// TwinCAT 3 PLC project PnP_MCgroupCM
// Title: Pick And Place Simple Example with MC Group Coordinated Motion
// Company: Beckhoff Automation GmbH
// Description: Disclaimer This publication contains statements about the suitability of our products for certain areas of application. These statements are based on typical features of our products. The examples shown in this publication are for demonstration purposes only. The information provided herein should not be regarded as specific operation characteristics. It is incumbent on the customer to check and decide whether a product is suitable for use in a particular application. We do not give any warranty that the source code which is made available with this publication is complete or accurate. THE SAMPLE CODE CONTAINED IN THIS PUBLICATION IS PROVIDED “AS IS” WITHOUT WARRANTY OF ANY KIND, EITHER EXPRESSED, IMPLIED OR STATUTORY, INCLUDING WITHOUT LIMITATION, ANY WARRANTY WITH RESPECT TO NON-INFRINGEMENT, FREEDOM FROM PROPRIETARY RIGHTS OF THIRD PARTIES OR FITNESS FOR ANY PARTICULAR PURPOSE. This publication may be changed from time to time without prior notice. No liability is assumed for errors and/or omissions. Our products are described in detail in our data sheets and documentations. Product-specific warnings and cautions must be observed. For the latest version of our data sheets and documentations visit our website (www.beckhoff.de). © Beckhoff Automation GmbH & Co. KG The reproduction, distribution and utilization of this document as well as the communication of its contents to others without express authorization is prohibited. Offenders will be held liable for the payment of damages. All rights reserved in the event of the grant of a patent, utility model or design.
// ProgramVersion: 3.1.4018.1
// libraries:
//   PLCToolbox, * (Beckhoff Automation LLC.)
//   Tc2_MC2, * (Beckhoff Automation GmbH)
//   Tc2_Standard, * (Beckhoff Automation GmbH)
//   Tc2_System, * (Beckhoff Automation GmbH)
//   Tc2_Utilities, * (Beckhoff Automation GmbH)
//   Tc3_EventLogger, * (Beckhoff Automation GmbH)
//   Tc3_McCoordinatedMotion, * (Beckhoff Automation GmbH)
//   Tc3_Module, * (Beckhoff Automation GmbH)
// project tree:
//   DUT/ ST_DwellTime.TcDUT, ST_LineSegment.TcDUT
//   / E_Axis.TcDUT, PlcTask.TcTTO
//   GVLs/ GVL.TcGVL
//   POUs/ FB_AddAllAxes.TcPOU, FB_PowerAll.TcPOU, FB_PreparePath.TcPOU, MAIN.TcPOU
// real-time tasks:
//   TASK PlcTask: cycle T#10ms, priority 20, ADS port 350
//   TASK Worker Task: cycle default, priority 32
// motion (NC):
//   TASK NC-Task 1 SAF: cycle T#2ms, priority 4, ADS port 501
//   TASK NC-Task 1 SVB: cycle T#10ms, priority 8, ADS port 511
//   AXIS X (id 1)
//     OtherSettings: AllowMotionCmdToSlave=true
//     encoder EncType=1
//     drive DrvType=5
//       TimeComp: TaskDelayCycles=1
//     controller CtrType=1
//       CtrPara: PriorControlFactor=1
//         Observer: BandWidth=20
//   AXIS Y (id 2)
//     OtherSettings: AllowMotionCmdToSlave=true
//     encoder EncType=1
//     drive DrvType=5
//       TimeComp: TaskDelayCycles=1
//     controller CtrType=1
//       CtrPara: PriorControlFactor=1
//         Observer: BandWidth=20
// variable links:
//   PnP_MCgroupCM/PnP_MCgroupCM Instance <-> NC-Task 1 SAF/Axes/X
//     PlcTask Inputs/GVL.stAxis[1].NcToPlc <-> Outputs/ToPlc
//     PlcTask Outputs/GVL.stAxis[1].PlcToNc <-> Inputs/FromPlc
//   PnP_MCgroupCM/PnP_MCgroupCM Instance <-> NC-Task 1 SAF/Axes/Y
//     PlcTask Inputs/GVL.stAxis[2].NcToPlc <-> Outputs/ToPlc
//     PlcTask Outputs/GVL.stAxis[2].PlcToNc <-> Inputs/FromPlc
//   PnP_MCgroupCM/PnP_MCgroupCM Instance <-> NC-Task 1 SAF/Objects/Group2 (MC Group Coordinated Motion)
//     PlcTask Inputs/GVL.stGroupRef.NcToPlc <-> Group Outputs/ToPLC
//     PlcTask Outputs/GVL.stGroupRef.PlcToNc <-> Group Inputs/FromPLC

CONFIGURATION PnP_MCgroupCM
    RESOURCE PLC ON TwinCAT3
        TASK PlcTask(INTERVAL := T#10ms, PRIORITY := 20);
        PROGRAM MAIN WITH PlcTask : MAIN;
    END_RESOURCE
END_CONFIGURATION

// ---- DUT/ST_DwellTime.TcDUT
TYPE ST_DwellTime :
STRUCT
	DwellTime	: TIME;
	BufferMode	: MC_BUFFER_MODE := mcBuffered;
	InvokeId	: UDINT;
END_STRUCT
END_TYPE

// ---- DUT/ST_LineSegment.TcDUT
TYPE
ST_LineSegment :
STRUCT
	TargetPos					: ARRAY[1..cAxesCount] OF MC_LREAL;
	Velocity					: MC_LREAL	:= MC_INVALID;
	Acceleration				: MC_LREAL	:= MC_DEFAULT;
	Deceleration				: MC_LREAL	:= MC_DEFAULT;
	Jerk						: MC_LREAL	:= MC_DEFAULT;
	TransitionParam				: ARRAY[1..2] OF MC_LREAL; //1 = blending distance on previous segment, defines when to leave line. 2 = blending distance on this segment, defines latest positionn to be back on line 
	BufferMode					: MC_BUFFER_MODE		:= MC_BUFFER_MODE.mcBlendingPrevious;
	TransitionMode				: MC_TRANSITION_MODE	:= MC_TRANSITION_MODE.mcTransModeCornerDistanceAdvanced;
	TransitionParameterCount	: UDINT					:= 2;
	InvokeId					: UDINT;
END_STRUCT
END_TYPE

// ---- E_Axis.TcDUT
{attribute 'qualified_only'}
{attribute 'strict'}
TYPE
E_Axis :
(
	X	:= 1,
	Y	:= 2,
	Z	:= 3
);
END_TYPE

// ---- GVLs/GVL.TcGVL
VAR_GLOBAL
	stGroupRef	: AXES_GROUP_REF;
	stAxis		: ARRAY[1..cAxesCount] OF AXIS_REF;
END_VAR

VAR_GLOBAL CONSTANT
	cAxesCount : UINT := 2;
END_VAR

// ---- POUs/MAIN.TcPOU
PROGRAM MAIN
VAR
	xInit	: BOOL := TRUE;
	fbMsg	: FB_TcMessage;
	Step	: (INIT,
		IDEL,
		ENABLE_AXIS,
		ADD_AXIS_TO_GROUP,
		ENABLE_GROUP,
		PREPARE_PATH,
		MOVE_PATH,
		WAIT_TILL_NO_MOVEMENT,
		UNGROUP_GROUP,
		STOPPING,
		ERROR,
		RESETING);

	Start, Stop, Reset	: BOOL;
	Continuous			: BOOL := TRUE;
	rtStart				: R_TRIG;
	rtReset				: R_TRIG;

	buffer	: ARRAY[1..4096] OF BYTE;
	path	: MC_PATH_DATA_REF(ADR(buffer), SIZEOF(buffer));

	fbPreparePath : FB_PreparePath;

	StartPos : ST_LineSegment := (TargetPos := [200.0, 275.0], Velocity := 500.0, TransitionParam := [2(0.0)], InvokeId := 10);

	Dwell : ST_DwellTime := (DwellTime := TIME#5S0MS, InvokeId := 15);

	Point1 : ST_LineSegment := (TargetPos					:= [279.0, 512],
								Velocity					:= 1600.0,
								Acceleration				:= 20000.0,
								Deceleration				:= 20000.0,
								Jerk						:= 60000.0,
								TransitionMode				:= MC_TRANSITION_MODE.mcTransModeCornerDistanceAdvanced,
								TransitionParam				:= [0.0, 0.0],
								TransitionParameterCount	:= 2,
								InvokeId					:= 20);

	Point2 : ST_LineSegment := (TargetPos					:= [417.0, 512.0],
								Velocity					:= 1160.0,
								Acceleration				:= 20000.0,
								Deceleration				:= 20000.0,
								Jerk						:= 60000.0,
								TransitionMode				:= MC_TRANSITION_MODE.mcTransModeCornerDistanceAdvanced,
								TransitionParam				:= [20.0, 25.0],
								TransitionParameterCount	:= 2,
								InvokeId					:= 30);

	fVelFactor : LREAL := 1.0;

	fbPower			: FB_PowerAll;
	fbAddAllAxes	: FB_AddAllAxes;
	fbGroupEnable	: MC_GroupEnable;

	fbMovePath			: MC_MovePath;
	fbStop				: MC_GroupStop;
	fbUngroupAxes		: MC_UngroupAllAxes;
	fbGroupReset		: MC_GroupReset;
	fbGroupReadStatus	: MC_GroupReadStatus;
	fbGroupSetOvr		: MC_GroupSetOverride;

END_VAR

IF xInit THEN
	xInit := FALSE;
	fbMsg.CreateEx(TC_EVENTS.Msg.Msg, 0);
	fbPreparePath(path := path);
END_IF

fbPower();

rtStart(CLK := Start);

CASE Step OF

	INIT:
		fbAddAllAxes(Execute := FALSE);
		fbGroupEnable(AxesGroup := stGroupRef, Execute := FALSE);
		fbMovePath(AxesGroup := stGroupRef, PathData := path, Execute := FALSE);
		Step := IDEL;

	IDEL:
		IF rtStart.Q THEN
			Step := ENABLE_AXIS;
		END_IF

	ENABLE_AXIS:
		fbPower.Enable := TRUE;

		IF fbPower.Status THEN
			Step := ADD_AXIS_TO_GROUP;
		ELSIF fbPower.Error THEN
			Step := ERROR;
			fbMsg.ipArguments.Clear();
			fbMsg.ipArguments.AddString('Error enabling axis');
			fbMsg.Send(0);
		END_IF

	ADD_AXIS_TO_GROUP:

		fbAddAllAxes(Execute := TRUE);

		IF fbAddAllAxes.Done THEN
			fbAddAllAxes(Execute := FALSE);
			Step := ENABLE_GROUP;
		ELSIF fbAddAllAxes.Error THEN
			Step := ERROR;
			fbMsg.ipArguments.Clear();
			fbMsg.ipArguments.AddString('Error adding axis to the group');
			fbMsg.Send(0);
		END_IF

	ENABLE_GROUP:

		fbGroupEnable(AxesGroup := stGroupRef, Execute := TRUE);

		IF fbGroupEnable.Done THEN
			fbGroupEnable(AxesGroup := stGroupRef, Execute := FALSE);
			Step := PREPARE_PATH;
		ELSIF fbGroupEnable.Error THEN
			Step := ERROR;
			fbMsg.ipArguments.Clear();
			fbMsg.ipArguments.AddString('Error: ').AddUDInt(fbGroupEnable.ErrorId).AddString(' enabling the group');
			fbMsg.Send(0);
		END_IF

	PREPARE_PATH:
		A_PreparePath();
		Step := MOVE_PATH;

	MOVE_PATH:

		fbMovePath(AxesGroup	:= stGroupRef,
					PathData	:= path,
					Execute		:= TRUE);

		IF fbMovePath.Done THEN
			fbMovePath(AxesGroup := stGroupRef, PathData := path, Execute := FALSE);
			Step := WAIT_TILL_NO_MOVEMENT;
		ELSIF fbMovePath.Error THEN
			Step := ERROR;
			fbMsg.ipArguments.Clear();
			fbMsg.ipArguments.AddString('Error: ').AddUDInt(fbMovePath.ErrorId).AddString(' on move path');
			fbMsg.Send(0);
		END_IF

	WAIT_TILL_NO_MOVEMENT:
		//Check that axes are not moving else we will get a position jump
		IF fbGroupReadStatus.GroupStandby OR fbGroupReadStatus.GroupErrorStop OR fbGroupReadStatus.GroupNotReady THEN
			fbUngroupAxes(AxesGroup := stGroupRef, Execute := FALSE);

			IF NOT Continuous THEN
				Step := UNGROUP_GROUP;
			ELSE
				Step := PREPARE_PATH;
			END_IF

		END_IF

	UNGROUP_GROUP:
		fbUngroupAxes(AxesGroup	:= stGroupRef,
						Execute	:= TRUE);

		IF fbUngroupAxes.Done THEN
			Step := IDEL;
		ELSIF fbUngroupAxes.Error THEN
			Step := ERROR;
			fbMsg.ipArguments.Clear();
			fbMsg.ipArguments.AddString('Error: ').AddUDInt(fbUngroupAxes.ErrorId).AddString(' on ungroup');
			fbMsg.Send(0);
		END_IF

	STOPPING:
		Stop := FALSE;
		fbStop(AxesGroup := stGroupRef, Execute := TRUE, Jerk := MC_IGNORE);

		IF fbStop.Done THEN
			fbStop(AxesGroup := stGroupRef, Execute := FALSE);
			Step := IDEL;
		ELSIF fbStop.Error THEN
			Step := ERROR;
			fbMsg.ipArguments.Clear();
			fbMsg.ipArguments.AddString('Error: ').AddUDInt(fbStop.ErrorId).AddString(' on stopping');
			fbMsg.Send(0);
		END_IF

	ERROR:
		IF rtReset.Q THEN
			Step := RESETING;
		END_IF

	RESETING:
		fbGroupReset(AxesGroup	:= stGroupRef,
					Execute		:= TRUE);

		IF fbGroupReset.Done THEN
			fbGroupReset(AxesGroup := stGroupRef, Execute := FALSE);

			IF fbGroupReadStatus.GroupDisabled THEN
				Step := IDEL;
			ELSE
				Step := INIT;
			END_IF
		END_IF
END_CASE

IF Stop AND Step <> STOPPING THEN
	Step := STOPPING;
END_IF

fbGroupReadStatus(AxesGroup := stGroupRef, Enable := TRUE);

IF fbGroupReadStatus.Error THEN
	Step := ERROR;
ELSIF NOT fbGroupReadStatus.Valid THEN
	Step := ERROR;
END_IF

fbGroupSetOvr(AxesGroup := stGroupRef, Enable := TRUE, VelFactor := fVelFactor);

IF fbGroupSetOvr.Error THEN
	Step := ERROR;
END_IF

ACTION A_PreparePath:
path.ClearPath(); //Clear nodes that were in path

//Start Position
fbPreparePath.AddLinearAbsolute(LineSegment := StartPos);

//Dwell
fbPreparePath.AddDwellTime(DwellTime := Dwell);

//Point 1
fbPreparePath.AddLinearAbsolute(LineSegment := Point1);

//Point 2
fbPreparePath.AddLinearAbsolute(LineSegment := Point2);
END_ACTION

END_PROGRAM

// ---- POUs/FB_PreparePath.TcPOU
FUNCTION_BLOCK FB_PreparePath
VAR_IN_OUT
	path : MC_PATH_DATA_REF;
END_VAR
VAR_OUTPUT
END_VAR
VAR

END_VAR

METHOD AddDwellTime : UDINT
VAR_INPUT
	DwellTime : ST_DwellTime;
END_VAR
VAR_INST
	fbDwellPrep	: MC_DwellTimePreparation;
	xInit		: BOOL := TRUE;
	fbMsg		: FB_TcMessage;
END_VAR
IF xInit THEN
	xInit := FALSE;
	fbMsg.CreateEx(TC_EVENTS.Msg.Msg, 0);
END_IF

fbDwellPrep(PathData	:= path,
			DwellTime	:= DwellTime.DwellTime,
			BufferMode	:= DwellTime.BufferMode,
			InvokeId	:= DwellTime.InvokeId);

IF fbDwellPrep.Error THEN
	fbMsg.ipArguments.Clear();
	fbMsg.ipArguments.AddString('Error: ').AddUDInt(fbDwellPrep.ErrorId).AddString(' on dwell prep').AddString('Invoke ID: ')
		.AddUDInt(fbDwellPrep.InvokeId);
END_IF

AddDwellTime := fbDwellPrep.ErrorId;
END_METHOD

METHOD AddLinearAbsolute : UDINT
VAR_INPUT
	LineSegment : ST_LineSegment;
END_VAR
VAR_INST
	fbMoveLinPrep	: MC_MoveLinearAbsolutePreparation;	
	xInit			: BOOL := TRUE;
	fbMsg			: FB_TcMessage;
END_VAR
IF xInit THEN
	xInit := FALSE;
	fbMsg.CreateEx(TC_EVENTS.Msg.Msg, 0);
END_IF

fbMoveLinPrep(PathData						:= path,
				Position					:= ADR(LineSegment.TargetPos),
				PositionCount				:= cAxesCount,
				Velocity					:= LineSegment.Velocity,
				Acceleration				:= LineSegment.Acceleration,
				Deceleration				:= LineSegment.Deceleration,
				Jerk						:= LineSegment.Jerk,
				BufferMode					:= LineSegment.BufferMode,
				TransitionMode				:= LineSegment.TransitionMode,
				TransitionParameter			:= ADR(LineSegment.TransitionParam),
				TransitionParameterCount	:= LineSegment.TransitionParameterCount,
				InvokeId					:= LineSegment.InvokeId);

IF fbMoveLinPrep.Error THEN
	fbMsg.ipArguments.Clear();
	fbMsg.ipArguments.AddString('Error: ').AddUDInt(fbMoveLinPrep.ErrorId).AddString(' on move line prep').AddString('Invoke ID: ')
		.AddUDInt(fbMoveLinPrep.InvokeId);
	fbMsg.Send(0);
END_IF

AddLinearAbsolute:=fbMoveLinPrep.ErrorId;
END_METHOD

END_FUNCTION_BLOCK

// ---- POUs/FB_PowerAll.TcPOU
FUNCTION_BLOCK FB_PowerAll
VAR_INPUT
	Enable : BOOL;
END_VAR
VAR_OUTPUT
	Status	: BOOL;
	Error	: BOOL;
END_VAR
VAR
	fbPower	: ARRAY[1..cAxesCount] OF MC_Power;
	i		: UINT;
END_VAR

Status	:= TRUE;
Error	:= FALSE;

FOR i := 1 TO cAxesCount DO
	fbPower[i](Axis				:= stAxis[i],
				Enable			:= Enable,
				Enable_Positive	:= Enable,
				Enable_Negative	:= Enable);

	Status	:= Status AND fbPower[i].Status;
	Error	:= Error OR fbPower[i].Error;
END_FOR

END_FUNCTION_BLOCK

// ---- POUs/FB_AddAllAxes.TcPOU
FUNCTION_BLOCK FB_AddAllAxes
VAR_INPUT
	Execute : BOOL;
END_VAR
VAR_OUTPUT
	Done	: BOOL;
	Busy	: BOOL;
	Error	: BOOL;
END_VAR
VAR
	fbAddAxis	: ARRAY[1..cAxesCount] OF MC_AddAxisToGroup;
	i			: UINT;
END_VAR

Done	:= TRUE;
Busy	:= FALSE;
Error	:= FALSE;

fbAddAxis[E_Axis.X].IdentInGroup	:= MCS_X;	//X-Axis
fbAddAxis[E_Axis.Y].IdentInGroup	:= MCS_Y;	//Y-Axis
//fbAddAxis[3].IdentInGroup := MCS_Z; //Z-Axis
//fbAddAxis[4].IdentInGroup := MCS_Z; //C-Axis

FOR i := 1 TO cAxesCount DO
	fbAddAxis[i](AxesGroup := stGroupRef, Axis := stAxis[i], Execute := Execute);

	IF (NOT fbAddAxis[i].Done) THEN
		Done := FALSE;
	END_IF

	IF (fbAddAxis[i].Busy) THEN
		Busy := TRUE;
	END_IF

	IF (fbAddAxis[i].Error) THEN
		Error := TRUE;
	END_IF
END_FOR

END_FUNCTION_BLOCK
